TYPE AdsSymbolUploadInfo :
STRUCT
   nSymbols : UDINT;
   nSymSize : UDINT;
END_STRUCT
END_TYPE

(* stored: Version 1.1.0.1, ProductVersion 3.1.4024.3
   DUT AdsSymbolUploadInfo: Id {88e2b59a-b2f9-4954-83ea-4fbe284a5635} *)
